FUNCTION_BLOCK FB_Sequencer
VAR CONSTANT
	NUM_MOTORS : INT := 5;
END_VAR
VAR
	
	Motors : ARRAY [1..NUM_MOTORS] OF Motor;
	MotorsI : ARRAY [1..NUM_MOTORS] OF MotorInputVariables;
	MotorsO : ARRAY [1..NUM_MOTORS] OF MotorOutputVariables;
	
	serialIndex : INT := 1;
	index : INT;
	
	generalStart : BOOL;
	generalStop : BOOL;
	resetFault : BOOL;
	
	stopTrig : R_TRIG;
	resetTrig : R_TRIG;
	
	SUCCEED: BOOL;
	FAIL: BOOL;
END_VAR

Ini_Motors();
mGeneralStop();
mFaultHandler();
mSequenceStart();

METHOD Ini_Motors : BOOL
VAR_INPUT
END_VAR
FOR index := 1 TO NUM_MOTORS BY 1 DO
	MotorsI[index].stop := generalStop;
	MotorsI[index].waitTime := T#2S;
	Motors[index](MotorInputs := MotorsI[index], MotorOutputs => MotorsO[index]);
END_FOR
END_METHOD

METHOD mFaultHandler : BOOL
VAR_INPUT
END_VAR
FOR index := 1 TO NUM_MOTORS BY 1 DO
	IF MotorsI[index].overload THEN
		FAIL := TRUE;
		EXIT;
	END_IF
END_FOR

IF FAIL THEN
	FOR index := 1 TO NUM_MOTORS BY 1 DO
		motorsI[index].start := FALSE;
		generalStop := TRUE;
	END_FOR
END_IF

resetTrig(CLK := resetFault);
IF resetTrig.Q THEN
	FAIL := FALSE;
	generalStop := FALSE;
END_IF
END_METHOD

METHOD mGeneralStop : BOOL
VAR_INPUT
END_VAR
stopTrig(CLK := generalStop);

IF  stopTrig.Q THEN
	SUCCEED := FALSE;
	FOR index := 1 TO NUM_MOTORS BY 1 DO
		MotorsI[index].start := FALSE;
	END_FOR
END_IF
END_METHOD

METHOD mSequenceStart : BOOL
VAR_INPUT
END_VAR
MotorsI[1].start := generalStart;

IF MotorsO[serialIndex].coil AND (NOT SUCCEED) AND NOT FAIL THEN
	IF serialIndex > NUM_MOTORS THEN
		serialIndex := 1;
	ELSE
		serialIndex := serialIndex + 1;
		MotorsI[serialIndex].start := TRUE;
	END_IF
END_IF

IF serialIndex - 1 = NUM_MOTORS THEN
	SUCCEED := TRUE;
	serialIndex := 1;
END_IF
END_METHOD

END_FUNCTION_BLOCK

(* stored: Version 1.1.0.1, ProductVersion 3.1.4024.12
   POU FB_Sequencer: Id {173e461d-9352-4021-ad5b-56f97cbeee87}, SpecialFunc None
   Method Ini_Motors: Id {3d1fec7d-dc23-422b-b4cc-783784f3787f}
   Method mFaultHandler: Id {966aa395-a523-433f-a0c1-03b4ba08fcff}
   Method mGeneralStop: Id {0481f4b0-2d57-49ae-9746-b885b04f77d9}
   Method mSequenceStart: Id {40fd3afa-ac07-4299-8241-2914e967e420} *)
